// TIA Portal V16 export
// export: Created 2021-09-08T12:46:12.0351878Z, ExportSetting WithDefaults, DisplayName Totally Integrated Automation Portal, DisplayVersion V16 Update 3, DisplayName TIA Portal Version Control Interface, DisplayVersion V16 Update 2, DisplayName TIA Portal Openness, DisplayVersion V16 Update 3, DisplayName TIA Portal Teamcenter Gateway, DisplayVersion V16, DisplayName STEP 7 Professional, DisplayVersion V16 Update 3, DisplayName STEP 7 Safety, DisplayVersion V16, DisplayName WinCC Advanced, DisplayVersion V16 Update 3
DATA_BLOCK "dtUzData"   // DB7
{ S7_Optimized_Access := 'FALSE' }
VERSION : 0.1
// stored: AutoNumber true, DBAccessibleFromOPCUA true, IsOnlyStoredInLoadMemory false, IsWriteProtectedInAS false
   VAR
      UZ30x : "UZ_Data";
      UZ901 { S7_SetPoint := 'True'} : "UZ_Data";
      UZ1301 { S7_SetPoint := 'True'} : "UZ_Data";
      UZ120x { S7_SetPoint := 'True'} : "UZ_Data";
      UZ150x { S7_SetPoint := 'True'} : "UZ_Data";
   END_VAR
BEGIN
END_DATA_BLOCK
